TYPE typeNewMsg :
STRUCT
	
timeRaised:STRING(12):='12:23:32';;
timeResolved:STRING(12):='13:43:12';
text:STRING(255);
source:STRING(10);


END_STRUCT
END_TYPE

(* stored: Version 1.1.0.1, ProductVersion 3.1.4024.12
   DUT typeNewMsg: Id {14c30d24-222e-4f0d-a8b9-6aa744ae4ded} *)
